PROGRAM p01_sequential
VAR
	S0 AT %I*: BOOL;
	S1 AT %I*: BOOL;
	L0 AT %Q*: BOOL;
	L1 AT %Q*: BOOL;
END_VAR

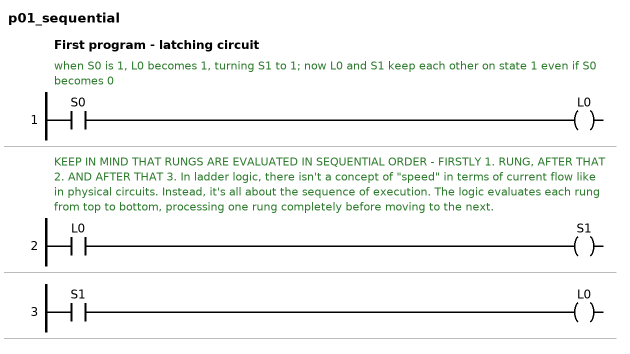
// NETWORK 1: First program - latching circuit
// when S0 is 1, L0 becomes 1, turning S1 to 1; now L0 and S1 keep each other on state 1 even if S0 becomes 0
L0 := S0;

// NETWORK 2
// KEEP IN MIND THAT RUNGS ARE EVALUATED IN SEQUENTIAL ORDER - FIRSTLY 1. RUNG, AFTER THAT 2. AND AFTER THAT 3. In ladder logic, there isn't a concept of "speed" in terms of current flow like in physical circuits. Instead, it's all about the sequence of execution. The logic evaluates each rung from top to bottom, processing one rung completely before moving to the next.
S1 := L0;

// NETWORK 3
L0 := S1;

END_PROGRAM

(* stored: Version 1.1.0.1, ProductVersion 3.1.4024.13
   POU p01_sequential: Id {6a847bd2-3fe6-4150-82aa-7c77e2c41670}, SpecialFunc None *)
